# EPICS IOC start-up script: iocsh/ethercatmcEL6688-PILS.iocsh
dbLoadRecords("ethercatmcEL6688-PILS.template", "PREFIX=$(PREFIX), MOTOR_PORT=$(MOTOR_PORT)")
